PROGRAM OP120_Robo_Inputs
VAR
	Robo_Enable_err: TON;
	temp : ARRAY[1..500] OF BOOL;
	
END_VAR




// Safe to Pick
IF OperationEnable AND OP120_GVL.CR120_Lifting_Cyl.Position2  THEN
	OP120_SI_Pick_Zone_Safe:=TRUE;
	ELSE
		OP120_SI_Pick_Zone_Safe:=FALSE;
	END_IF
	
// Safe To Place
IF OperationEnable AND OP120_GVL.CR120_Horizontal_Push_Cyl.Position1 THEN
	OP120_IO_Tag_Link.OP120_SI_Place_Zone_Safe:=TRUE;
	ELSE
		OP120_IO_Tag_Link.OP120_SI_Place_Zone_Safe:=FALSE;
	END_IF
//Safe to Reject Zone
	
	IF OperationEnable AND TRUE THEN
		OP120_IO_Tag_Link.OP120_SI_Reject_Zone_Safe:=TRUE;
		ELSE
			OP120_IO_Tag_Link.OP120_SI_Reject_Zone_Safe:=FALSE;
		END_IF
// Safe to ATC Zone
IF OperationEnable THEN
	OP120_IO_Tag_Link.OP120_SI_ATC_Tool_Safe:=TRUE;
	ELSE
	OP120_IO_Tag_Link.OP120_SI_ATC_Tool_Safe:=FALSE;
	END_IF

//Ready to Pick
IF OP120_GVL.OP120_StartEnable AND OP120_GVL.CR120_Lifting_Cyl.Position2 AND OP120_GotoPick THEN 
	// AND CheckParkOK AND NOT  CheckParkNOK and (OP120_EI_Gripper1_Open AND  OP120_EI_Gripper2_Open OR temp [1])
   OP120_EI_Rdy_Pick_Spring :=TRUE;
ELSE
	OP120_IO_Tag_Link.OP120_EI_Rdy_Pick_Spring :=FALSE;
END_IF 

//REady to 	place

IF OP120_GVL.OP120_StartEnable AND OP120_GVL.CR120_Horizontal_Push_Cyl.Position1 AND OP120_MoverPresent  THEN //OP120_STN_ENABLE AND Part_Picked
	OP120_IO_Tag_Link.OP120_EI_Rdy_Place_Spring:=TRUE;
	ELSE
	OP120_IO_Tag_Link.OP120_EI_Rdy_Place_Spring:=FALSE;
END_IF

//Insertion Complete

IF OP120_GVL.OP120_StartEnable AND OP120_PartPushed THEN
	OP120_IO_Tag_Link.OP120_EI_Insertion_Complete:=TRUE;
ELSE
	OP120_IO_Tag_Link.OP120_EI_Insertion_Complete:=FALSE;
END_IF

END_PROGRAM

(* stored: Version 1.1.0.1, ProductVersion 3.1.4024.11
   POU OP120_Robo_Inputs: Id {77b19724-6ce1-4629-b652-37b54d0adf57}, SpecialFunc None *)
